// TIA Portal project "Groups" (V15.1)

(* hardware
DEVICE "S71500/ET200MP station_1"  S7-1500 station
   slot 0: "Rail_0"  Rack  6ES7 590-1***0-0AA0
   slot 1: "-PLC"  CPU 1515F-2 PN  6ES7 515-2FM01-0AB0  V2.6
      slot 3: "CPU display_1"  6ES7591-1BA00-0AA0
   slot 2: "F-DI 16x24V DC_1"  F-DI 16x24V DC  6ES7 526-1BH00-0AB0  V1.0
      slot 1: "F-DI 16x24V DC_1"  F-DI 16x24V DC
   slot 3: "F-DQ 8x24V DC/2A PPM_1"  F-DQ 8x24V DC/2A PPM  6ES7 526-2BF00-0AB0  V1.0
      slot 1: "F-DQ 8x24V DC/2A PPM_1"  F-DQ 8x24V DC/2A PPM
DEVICE "HMI_1"  TP900 Comfort
   slot 0: "HMI"  TP900 Comfort  6AV2 124-0JC01-0AX0  15.1.0.0
   slot 1: "HMI_RT_1"  TP900 Comfort  6AV2 124-0JC01-0AX0  15.1.0.0
   slot 5: "HMI._CP_1"  PROFINET Interface  15.0.1.0
      slot 1: "PROFINET Interface_1"  PROFINET Interface
         slot 1: "hmi_Port_1"  Port
         slot 2: "hmi_Port_2"  Port
   slot 7: "HMI.I/DP_CP_1"  MPI/DP Interface  15.0.1.0
DEVICE "SINAMICS G_1"  Sinamics.Device
   slot 0: "	_0"  Rail  SinamicsG120RackPN
   slot 0: "-Drive"  G120 CU240E-2 PN-F  6SL3244-0BB13-1FA0  4.7.10
      slot 1: "PROFINET interface"  MDD-SinamicsG120-P
   slot 3: "PM240-2 IP20"  PM240-2 IP20  6SL3210-1PE12-3ULx  -
DEVICE "S71500/ET200MP station_2"  S7-1500 station
   slot 0: "Rail_0"  Rack  6ES7 590-1***0-0AA0
   slot 1: "TC"  CPU 1518F-4 PN/DP  6ES7 518-4FP00-0AB0  V2.6
      slot 3: "CPU display_1"  6ES7591-1BA00-0AA0
DEVICE "SCALANCE W client"  SCALANCE W-Station
   slot 0: "SCALANCE W rack"  Rail
   slot 0: "-WLAN"  SCALANCE W734-1 RJ45 US  6GK5 734-1FX00-0AB0  V6.2
DEVICE "ET 200SP station_1"  ET 200SP-Station
   slot 0: "Rack_0"  Rack  6ES5 710-8MAx1
   slot 0: "-IO device_1"  IM 155-6 PN/2 HF  6ES7 155-6AU01-0CN0  V4.2
   slot 1: "DI 8x24VDC HF_1"  DI 8x24VDC HF  6ES7 131-6BF00-0CA0  V2.0
      slot 1: "DI 8x24VDC HF_1"  DI 8x24VDC HF
   slot 2: "F-DI 8x24VDC HF_1"  F-DI 8x24VDC HF  6ES7 136-6BA00-0CA0  V1.0
      slot 1: "F-DI 8x24VDC HF_1"  F-DI 8x24VDC HF
   slot 3: "F-DQ 4x24VDC/2A PM HF_1"  F-DQ 4x24VDC/2A PM HF  6ES7 136-6DB00-0CA0  V2.0
      slot 1: "F-DQ 4x24VDC/2A PM HF_1"  F-DQ 4x24VDC/2A PM HF
   slot 4: "Server module_1"  Server module  6ES7 193-6PA00-0AA0  V1.1
      slot 1: "Server module_1"  Server module
   slot 127: "BA 2xRJ45"  BA 2xRJ45  6ES7 193-6AR00-0AA0  V0.0
      slot 1: "Port_1"  X1 P1 R  6ES7 193-6AR00-0AA0  V0.0
      slot 2: "Port_2"  X1 P2 R  6ES7 193-6AR00-0AA0  V0.0
DEVICE "ET200Pro station_1"  ET200Pro station
   slot 0: "Rack_0"  Rail
   slot 0: "-IO device_3"  IM 154-4 PN HF  6ES7 154-4AB10-0AB0  V7.1
   slot 2: "4/8 F-DI 4 F-DO_1"  4/8 F-DI 4 F-DO  6ES7 148-4FC00-0AB0
   slot 3: "F-Switch_1"  F-Switch  6ES7 148-4FS00-0AB0
   slot 4: "4DO x 24VDC / 2A_1"  4DO x 24VDC / 2A  6ES7 142-4BD00-0AA0
DEVICE "GSD device_15"  GSD.Device.PN
   slot 0: "Rack"  Rack  V1.0
   slot 0: "-ird400"  IRD400  6ES7 292-0AA50-1AA0  V01.00.02
      slot 0: "IRD400"  IRD400
      slot 1: "PNIO"  PNIO
         slot 1: "Port 1"  Port 1
         slot 2: "Port 2"  Port 2
      slot 1: "IR Remote Control"  IR Remote Control
         slot 0: "IR Remote Control"  IR Remote Control
      slot 2: "Display and LED"  Display and LED 
         slot 0: "Display and LED"  Display and LED 
      slot 3: "DIO"  DIO
         slot 0: "DIO"  DIO
      slot 4: "IR-P2P"  IR-P2P
         slot 0: "IR-P2P"  IR-P2P
      slot 5: "Device Control"  Device Control
         slot 0: "Device Control"  Device Control
DEVICE "GSD device_16"  GSD.Device.PN
   slot 0: "Rack"  Rack  V1.0
   slot 0: "-enc"  ENA58IL-MT1213  ENA58IL-PROFINET  V10.0
      slot 0: "DeviceItemData"  DAP3_STD_PDEV_MT1213
      slot 1: "PN-IO"  PN-IO
         slot 1: "Port 1"  Port 1
         slot 2: "Port 2"  Port 2
      slot 1: "Encoder Multiturn 25 Bit_1"  Encoder Multiturn 25 Bit
         slot 0: "Module Access Point"  Module Access Point
   slot 1: "Standard Telegram 83, PZD2/8"  Standard Telegram 83, PZD2/8
DEVICE "GSD device_1"  GSD.Device.PN
   slot 0: "Rack"  Rack  V1.0
   slot 0: "-rf180c"  RF180C V2.2  6GT2 002-0JD00  2.0
      slot 0: "Standard"  Standard
      slot 1: "RF180C Interface"  RF180C Interface
         slot 1: "Port 1"  Port 1
         slot 2: "Port 2"  Port 2
      slot 1: "2x RS422 channels RFID_1"  2x RS422 channels RFID
         slot 0: "2x RS422 channels RFID"  2x RS422 channels RFID
DEVICE "SCALANCE XC-200"  SCALANCE X-Station
   slot 0: "SCALANCE X rack"  Rail
   slot 0: "-Switch1"  SCALANCE XC208  6GK5 208-0BA00-2AC2  V4.0
DEVICE "ET 200SP station_2"  ET 200SP-Station
   slot 0: "Rack_0"  Rack  6ES5 710-8MAx1
   slot 0: "-IO device_2"  IM 155-6 PN/2 HF  6ES7 155-6AU01-0CN0  V4.2
   slot 1: "DI 8x24VDC HF_1"  DI 8x24VDC HF  6ES7 131-6BF00-0CA0  V2.0
      slot 1: "DI 8x24VDC HF_1"  DI 8x24VDC HF
   slot 2: "F-DI 8x24VDC HF_1"  F-DI 8x24VDC HF  6ES7 136-6BA00-0CA0  V1.0
      slot 1: "F-DI 8x24VDC HF_1"  F-DI 8x24VDC HF
   slot 3: "F-DQ 4x24VDC/2A PM HF_1"  F-DQ 4x24VDC/2A PM HF  6ES7 136-6DB00-0CA0  V2.0
      slot 1: "F-DQ 4x24VDC/2A PM HF_1"  F-DQ 4x24VDC/2A PM HF
   slot 4: "Server module_1"  Server module  6ES7 193-6PA00-0AA0  V1.1
      slot 1: "Server module_1"  Server module
   slot 127: "BA 2xRJ45"  BA 2xRJ45  6ES7 193-6AR00-0AA0  V0.0
      slot 1: "Port_1"  X1 P1 R  6ES7 193-6AR00-0AA0  V0.0
      slot 2: "Port_2"  X1 P2 R  6ES7 193-6AR00-0AA0  V0.0
DEVICE "SCALANCE X-200"  SCALANCE X-Station
   slot 0: "SCALANCE X rack"  Rail
   slot 0: "Switch_2"  SCALANCE X208  6GK5 208-0BA10-2AA3  V5.2
*)

// ===== PLC "-PLC"  CPU 1515F-2 PN =====

VAR_GLOBAL   // PLC tag table "Default tag table"
   "Tag_1" AT %I56.1 : Bool;
   "Tag_2" AT %Q55.1 : Bool;
   "Tag_3" AT %I200.0 : Bool;
   "Tag_4" AT %Q200.0 : Bool;
   "Tag_5" AT %I56.0 : Bool;
   "Tag_6" AT %Q60.0 : Bool;
   "Tag_7" AT %I60.0 : Bool;
   "SpeedAxis_1_Actor_Interface_AddressIn" AT %I260.0 : "PD_TEL1_IN";
   "SpeedAxis_1_Actor_Interface_AddressOut" AT %Q260.0 : "PD_TEL1_OUT";
   "RopeEncoder_Sensor_Interface_AddressIn" AT %I316.0 : "PD_TEL83_IN";
   "RopeEncoder_Sensor_Interface_AddressOut" AT %Q304.0 : "PD_TEL83_OUT";
END_VAR

DATA_BLOCK "Main_Safety_RTG1_DB"   // DB1, F_DB
{ S7_Optimized_Access := 'TRUE' }
NAME : FUSI
VERSION : 0.1
// stored: InstanceOfName Main_Safety_RTG1
"Main_Safety_RTG1"
BEGIN
END_DATA_BLOCK

DATA_BLOCK "SpeedAxis_1"   // DB2, Motion_DB
{ S7_Optimized_Access := 'TRUE' }
AUTHOR : SIMATIC
FAMILY : MC_1500
VERSION : 4.0
// stored: InstanceOfName TO_SpeedAxis
"TO_SpeedAxis"
BEGIN
END_DATA_BLOCK

DATA_BLOCK "SIMATIC Ident_1"   // DB30
{ S7_Optimized_Access := 'TRUE' }
AUTHOR : SIMATIC
FAMILY : Ident
VERSION : 1.0
// stored: InstanceOfName TO_IDENT
"TO_IDENT"
BEGIN
   LADDR := 16#003C;
   HW_ID := 16#0134;
   CM_CHANNEL := 1;
END_DATA_BLOCK

DATA_BLOCK "RopeEncoder"   // DB2001, Motion_DB
{ S7_Optimized_Access := 'TRUE' }
AUTHOR : SIMATIC
FAMILY : MC_1500
VERSION : 4.0
// stored: InstanceOfName TO_ExternalEncoder
"TO_ExternalEncoder"
BEGIN
END_DATA_BLOCK

FUNCTION_BLOCK "Main_Safety_RTG1"   // FB1, F_LAD
{ S7_Optimized_Access := 'TRUE' }
VERSION : 0.1
BEGIN

REGION Network 1
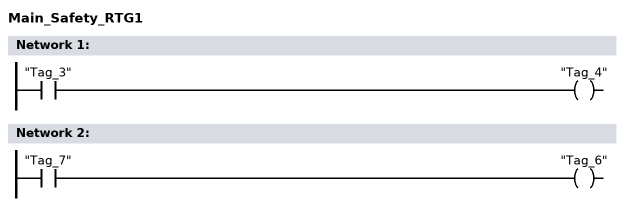
   RUNG wire#powerrail
      Contact( "Tag_3" )
      Coil( "Tag_4" )
   END_RUNG
   // the same network as SCL:
   "Tag_4" := "Tag_3";
END_REGION

REGION Network 2
   RUNG wire#powerrail
      Contact( "Tag_7" )
      Coil( "Tag_6" )
   END_RUNG
   // the same network as SCL:
   "Tag_6" := "Tag_7";
END_REGION
END_FUNCTION_BLOCK

FUNCTION "FC_Block_1" : Void   // FC1, LAD
{ S7_Optimized_Access := 'TRUE' }
VERSION : 0.1
   VAR_INPUT
      in1 : Bool;
   END_VAR
   VAR_OUTPUT
      out1 : Bool;
   END_VAR
BEGIN

REGION Network 1
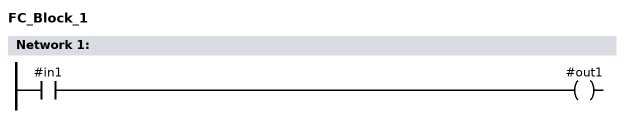
   RUNG wire#powerrail
      Contact( #in1 )
      Coil( #out1 )
   END_RUNG
   // the same network as SCL:
   #out1 := #in1;
END_REGION
END_FUNCTION

ORGANIZATION_BLOCK "Main"   // OB1, LAD, ProgramCycle
TITLE = "Main Program Sweep (Cycle)"
{ S7_Optimized_Access := 'TRUE' }
VERSION : 0.1
   VAR_INPUT
      Initial_Call : Bool;   // Initial call of this OB
      Remanence : Bool;   // =True, if remanent data are available
   END_VAR
BEGIN

REGION Network 1
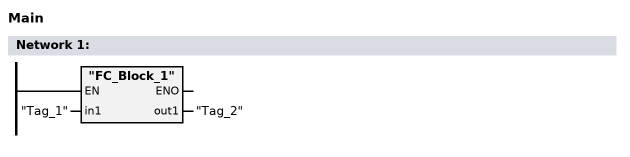
   RUNG wire#powerrail
      "FC_Block_1"(in1 := "Tag_1", out1 => "Tag_2")
   END_RUNG
   // the same network as SCL:
   "FC_Block_1"(in1 := "Tag_1", out1 => "Tag_2");
END_REGION
END_ORGANIZATION_BLOCK

// ===== PLC "TC"  CPU 1518F-4 PN/DP =====

DATA_BLOCK "Main_Safety_RTG1_DB"   // DB1, F_DB
{ S7_Optimized_Access := 'TRUE' }
NAME : FUSI
VERSION : 0.1
// stored: InstanceOfName Main_Safety_RTG1
"Main_Safety_RTG1"
BEGIN
END_DATA_BLOCK

FUNCTION_BLOCK "Main_Safety_RTG1"   // FB1, F_FBD
{ S7_Optimized_Access := 'TRUE' }
VERSION : 0.1
BEGIN
END_FUNCTION_BLOCK

ORGANIZATION_BLOCK "Main"   // OB1, LAD, ProgramCycle
TITLE = "Main Program Sweep (Cycle)"
{ S7_Optimized_Access := 'TRUE' }
VERSION : 0.1
   VAR_INPUT
      Initial_Call : Bool;   // Initial call of this OB
      Remanence : Bool;   // =True, if remanent data are available
   END_VAR
BEGIN
END_ORGANIZATION_BLOCK

(* ===== HMI "HMI_RT_1" =====
system functions are stored by id; their names below are inferred from use
connection "HMI_Connection_1": ETHERNET, S7_1500_OMS

HMI tags "Default tag table"
   "Tag_5" : Bool = PLC Tag_5 AT %I56.0, 1 s

screen "Screen_1" 800x480
   Button "Button_1" at 116,263 size 192x32; TextOff 'Screen_2'
      on Click: ActivateScreen("Screen_2", 0)
   IOField "I/O field_1" at 103,73 size 96x32; FormatPattern 1
      ProcessValue <- "Tag_5"
*)